TYPE ST_MachineStation :
STRUCT
	iSensorInfeed1, 		
	iSensorInfeed2, 		
	iSensorOutfeed1, 	
	iSensorOutfeed2, 	
	bButtonMachineStart,
	bButtonMachineStop,
	bButtonMachineReset : BOOL;
			
END_STRUCT
END_TYPE

(* stored: Version 1.1.0.1, ProductVersion 3.1.4024.12
   DUT ST_MachineStation: Id {2f0e25d1-d37d-4f19-bd82-514da3a27a02} *)
